// TIA Portal V21 export
VAR_GLOBAL   // PLC tag table "K_Fronte"
END_VAR
VAR_GLOBAL CONSTANT   // user constants
   K_Fronte_UtenzeInLavaggio : Int := 1;
END_VAR
